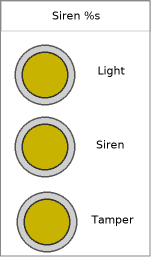
VISUALIZATION Siren  // 151x257
VAR_IN_OUT
	stSiren		: ST_AlarmSirenHMI;
END_VAR
    Lamp1 (10,40 70x70), variable: stSiren.bLight, style: Lamp-Lamp1-Yellow
    Lamp1 (10,112 70x70), variable: stSiren.bSiren, style: Lamp-Lamp1-Yellow
    Label (87,56 49x30), "Light"
    Label (86,130 49x30), "Siren"
    Textfield (1,1 150x30), "Siren %s", text variable: stSiren.sName
    Lamp1 (12,187 70x70), variable: stSiren.bTamper, style: Lamp-Lamp1-Yellow
    Label (88,205 49x30), "Tamper"
END_VISUALIZATION

(* stored: Version 1.1.0.1, ProductVersion 3.1.4024.12
   Visu Siren: Id {68fcba02-bdf0-4588-9545-5f238688fbe9} *)
